(* CODESYS project vacuumsystemsimulator.library
   Title: Vacuum System Simulator Library
   Description: Library of functions used for simulation of vacuum systems.
   Placeholder: Vacuum System Simulator Library
   Version: 0.2.10
   Company: SLAC

Project tree, tasks and I/O mapping:
  libraries: Tc2_ControllerToolbox, * (Beckhoff Automation GmbH); Tc2_Standard, * (Beckhoff Automation GmbH); Tc2_System, * (Beckhoff Automation GmbH); Tc3_Interfaces, * (Beckhoff Automation GmbH); Tc3_Module, * (Beckhoff Automation GmbH)
  DUTs/
    data type ST_CapManometer
    data type ST_CapManometer_CMR362
    data type ST_GAM_PIP
    data type ST_MechPump
    data type ST_MKS_275
    data type ST_MKS_317
    data type ST_MKS_422
    data type ST_MKS_500
    data type ST_MKS_626
    data type ST_MKS_722
    data type ST_MKS_903
    data type ST_MKS_907
    data type ST_MKS_909
    data type ST_MKS_925
    data type ST_TwinScrewRoughPump
    data type ST_VacuumGauge
    data type ST_VacuumValve
    data type ST_VAT_77FS
    data type ST_Volume
  GVLs/
    global variables GVL
    global variables GVL_VSS_CONSTANT
  POUs/
    VacuumGaugePressureFunctions/
      function F_MKS_937 [ST]
    function block FB_Aperture [ST]
    function block FB_CapManometer [ST]: M_CapManometer
    function block FB_CapManometer_CMR362 [ST]: M_CapManometer_CMR362
    function block FB_GAM_PIP [ST]
    function block FB_MKS_275 [ST]
    function block FB_MKS_275_to_500_HvOn [ST]
    function block FB_MKS_422 [ST]
    function block FB_MKS_500 [ST]: M_MKS_500
    function block FB_MKS_903 [ST]: M_MKS_903
    function block FB_MKS_907 [ST]: M_MKS_907
    function block FB_MKS_909 [ST]: M_MKS_909
    function block FB_MKS_925 [ST]: M_MKS_925
    function block FB_RoughPump [ST]
    function block FB_SetChamberPressure [ST]
    function block FB_TurboPump [ST]: PumpLogic
    function block FB_VacuumValve [ST]
    function block FB_VacuumValve_Vent [ST]
    function block FB_VirtualLeak [ST]
  Version/
    global variables Global_Version
  VISUs/
*)

// DUTs/ST_CapManometer
TYPE ST_CapManometer EXTENDS ST_VacuumGauge :
STRUCT
	//rFull_Scale used for scaling the voltage range of Capacitance
	//Manometer
	rFull_Scale : REAL; //in Torr
END_STRUCT
END_TYPE

// DUTs/ST_CapManometer_CMR362
TYPE ST_CapManometer_CMR362 EXTENDS ST_VacuumGauge :
STRUCT
	(*ST_CapManometer_CMR362 is a special CapManometer with a 
	rFull_Scale = 75.0 Torr*)
	
	//rFull_Scale used for scaling the voltage range of Capacitance
	//Manometer 
	rFull_Scale : REAL := 75.0 ;// Torr
END_STRUCT
END_TYPE

// DUTs/ST_GAM_PIP
TYPE ST_GAM_PIP :
STRUCT
	//Discrete Readback 
	xOn AT%I*:BOOL; //Readback of whether Gamma Ion Pump is turned on or not
END_STRUCT
END_TYPE

// DUTs/ST_MechPump
TYPE ST_MechPump :
STRUCT
	//Simulation Parameters
	rMRE	:	REAL; // Mass Removal Efficiency: should be a number less than 1.
	rBasePress	:	REAL := 1E-3;
	rLoad	:	REAL;
	iMaxSpd	:	INT;
	rMaxLoad	:	REAL;
	tonSpd	:	TON;
	tonTemp	:	TON;
	tonOvrLd	:	TON;
	xCooling:	BOOL := FALSE; // hook the cooling active signal here
	srError	:	SR;
	rtResetErr : R_TRIG;
	
	
	//Discrete controls
	i_xIlk	:	BOOL;//allow pump to turn on
	i_xRun	:	BOOL;//actually turn on pump
	
	//Discrete readbacks
	q_xAtSpd	:	BOOL;//whether pump is at top speed
	q_xErr	:	BOOL;//whether pump has an error or faulted
	q_xStart	:	BOOL;//whether pump has started but hasnt reached top speed, returns false when reaches top speeds
	q_xLowSpd	: BOOL;//whether pump is in a lowspeed STATE
	
	//Other Readbacks
	q_iPower	:	INT;
	q_iSpeed	:	INT;
END_STRUCT
END_TYPE

// DUTs/ST_MKS_275
TYPE ST_MKS_275 EXTENDS ST_VacuumGauge :
STRUCT
	stIntrpParams	:	ST_CTRL_LIN_INTERPOLATION_PARAMS;//setup for interpolating the Pirani's funky voltage to pressure transformation
	fbInterpolator	:	FB_CTRL_LIN_INTERPOLATION := (
		bExtrapolate := TRUE //can be false too
		);
END_STRUCT
END_TYPE

// DUTs/ST_MKS_317
TYPE ST_MKS_317 EXTENDS ST_VacuumGauge :
STRUCT
END_STRUCT
END_TYPE

// DUTs/ST_MKS_422
TYPE ST_MKS_422 EXTENDS ST_VacuumGauge :
STRUCT
	
	//Discrete Control: Ion gauges only
	i_xHvOn	 AT%I*:	BOOL;//High voltage On to turn on ion gauges
	
	// Simulation parameters
	tonIC	:	TON := (PT := T#10S);// takes 10 seconds to turn on this gauge
END_STRUCT
END_TYPE

// DUTs/ST_MKS_500
TYPE ST_MKS_500 EXTENDS ST_VacuumGauge :
STRUCT
	//Discrete Control: Ion gauges only
	i_xHvOn	 AT%I*:BOOL	; //High voltage On to turn on this Cold Cathode gauge
	q_xHVOn AT%Q*:BOOL ;
	q_DisActive AT%Q*:BOOL ;
	// Simulation parameters
	tonIC	:	TON := (PT := T#10S);// takes 10 seconds to turn on this Cold Cathode gauge
END_STRUCT
END_TYPE

// DUTs/ST_MKS_626
TYPE ST_MKS_626 EXTENDS ST_VacuumGauge :
STRUCT
END_STRUCT
END_TYPE

// DUTs/ST_MKS_722
TYPE ST_MKS_722 EXTENDS ST_VacuumGauge :
STRUCT
END_STRUCT
END_TYPE

// DUTs/ST_MKS_903
TYPE ST_MKS_903 EXTENDS ST_VacuumGauge:
STRUCT

	//Discrete Control: Ion gauges only
	i_xHvOn	:	BOOL;//High voltage On to turn on this Cold Cathode gauge
	
	// Simulation parameters
	tonIC	:	TON := (PT := T#10S);// takes 10 seconds to turn on this Cold Cathode gauge

END_STRUCT
END_TYPE

// DUTs/ST_MKS_907
TYPE ST_MKS_907 EXTENDS ST_VacuumGauge :
STRUCT
	stIntrpParams	:	ST_CTRL_LIN_INTERPOLATION_PARAMS;//setup for interpolating the Pirani's funky voltage to pressure transformation
	fbInterpolator	:	FB_CTRL_LIN_INTERPOLATION := (
		bExtrapolate := FALSE
);
END_STRUCT
END_TYPE

// DUTs/ST_MKS_909
TYPE ST_MKS_909 EXTENDS ST_VacuumGauge:
STRUCT

	//Discrete Control: Ion gauges only
	i_xHvOn	:	BOOL;//High voltage On to turn on this Hot Cathode gauge, they turn on immediately, unlike cold cathodes
	
END_STRUCT
END_TYPE

// DUTs/ST_MKS_925
TYPE ST_MKS_925 EXTENDS ST_VacuumGauge :
STRUCT
END_STRUCT
END_TYPE

// DUTs/ST_TwinScrewRoughPump
TYPE ST_TwinScrewRoughPump EXTENDS ST_MechPump :
STRUCT
	//Control
	i_xLowSpd	:	BOOL;
	i_xReset	:	BOOL;
	
	//Readback
	q_xRun		:	BOOL;
	q_xStop		:	BOOL;
	
END_STRUCT
END_TYPE

// DUTs/ST_VacuumGauge
TYPE ST_VacuumGauge :
STRUCT
	(* Simulation parameters *)
	rPress	:	REAL;//The real pressure coming from the ST_volume @ a chamber
	
	(* IO Readback *)
	q_iRawPress	 AT%Q*:	INT;// The transformed integer from real pressure to an integer encoded signal to be passed to the PLC 
	
	(* Testing Connection *)
	q_xGaugeConnected	: BOOL;// to connect and disconnect gauge, easy to check whether gauge in connected at correct location

END_STRUCT
END_TYPE

// DUTs/ST_VacuumValve
TYPE ST_VacuumValve :
STRUCT

	//Discrete controls
	i_xSol	 AT%I*	:BOOL;//Solenoid to control the valve( either closed or open)
	
	//Discrete readbacks
	q_xOpnLS  AT%Q*: BOOL;//readback whether open
	q_xClsLS  AT%Q*: BOOL;//readback whether closed
END_STRUCT
END_TYPE

// DUTs/ST_VAT_77FS
TYPE ST_VAT_77FS :
STRUCT
	(*HV sensor 1*)
	q_xSens1Rdy	:	BOOL;
	q_xSens1Inrush	:	BOOL;
	i_xSens1SensorOff:	BOOL;
	
	(*HV sensor 2*)
	q_xSens2Rdy	:	BOOL;
	q_xSens2Inrush	:	BOOL;
	i_xSens2SensorOff:	BOOL;
	
	(*Control Module*)
	q_xSysRdy	:	BOOL;
	q_xClsExternal	:	BOOL;
	i_xSysReset	:	BOOL;
	
	(*Gate Module*)
	q_xGate1Open:	BOOL;
	q_xGate1Close	:	BOOL;
	q_xGate1Rdy	:	BOOL;
	
	q_xGate2Open:	BOOL;
	q_xGate2Close	:	BOOL;
	q_xGate2Rdy	:	BOOL;
	
	i_xGate1Open:	BOOL;
	i_xGate1Close	:	BOOL;
	i_xGate2Open:	BOOL;
	i_xGate2Close	:	BOOL;
	
	(*FAST Shutter Valve Module*)
	q_xFast1Rdy	:	BOOL;
	q_xFast1Inrush	:	BOOL;
	i_xFast1SensorOff:	BOOL;
	
	i_xFast1Open:	BOOL;
	i_xFast1Close	:	BOOL;

END_STRUCT
END_TYPE

// DUTs/ST_Volume
TYPE ST_Volume :
STRUCT
	(*The Volume, Pressure, and LeakRate in each chamber
	Each chamber is divided up based on the one of the pages in the drawings*)
	rVolume : REAL;	
	rPressure : REAL; //in Torr
	rVLeak	:	REAL; //Torr*L/cycle
END_STRUCT
END_TYPE

// GVLs/GVL
VAR_GLOBAL
END_VAR

// GVLs/GVL_VSS_CONSTANT
VAR_GLOBAL CONSTANT
	ATM	:	REAL := 760; // Atmospheric pressure in Torr
	tSec : INT := 1; // time in seconds
	IonMassRate : REAL := 0.00001; // Torr*Liter/seconds
END_VAR

// Version/Global_Version
{attribute 'TcGenerated'}
// This function has been automatically generated from the project information.
VAR_GLOBAL CONSTANT
	{attribute 'const_non_replaced'}
	{attribute 'linkalways'}
	stLibVersion_Vacuum_System_Simulator_Library : ST_LibVersion := (iMajor := 0, iMinor := 2, iBuild := 10, iRevision := 0, sVersion := '0.2.10');
END_VAR

// POUs/VacuumGaugePressureFunctions/F_MKS_937
FUNCTION F_MKS_937 : INT
VAR_INPUT
	rPress	:	REAL;
END_VAR
VAR
END_VAR

(* Converts real pressure to digital voltage for 937A/B *)
IF rPress <> 0 THEN
	F_MKS_937 := REAL_TO_INT( (32767/10) * (0.6* LOG( rPress ) + 7.2) );
ELSE
	F_MKS_937 := 0;
END_IF

END_FUNCTION

// POUs/FB_Aperture
FUNCTION_BLOCK FB_Aperture
VAR_INPUT
	i_rC	:	REAL := 0.5; //Conductance (less than 1)
END_VAR
VAR_OUTPUT
END_VAR
VAR_IN_OUT
	stAVol	:	ST_Volume;
	stBVol	:	ST_Volume;
END_VAR
VAR
	Pa, Va, Pb, Vb	:	REAL;
	//DeltaPa, DeltaPb	:	REAL;
END_VAR

(* Aperture Simulation
A.Pai
3/29/2017

An aperture is like a valve that is permanently open but allows a restricted
amount of mass to flow through it. It has no polarity, that is to say,
it flows the same in either direction.

An aperture is the interface between two chambers and imitates the realistic
flow rate to adjust for changing pressures
*)

// Mass flow is dependent upon pressure differential, mass flow limited by aperture size.

Pa := stAVol.rPressure;
Va := stAVol.rVolume;

Pb := stBVol.rPressure;
Vb := stBVol.rVolume;

(*simplified version of Mass in chamber = old mass - mass flow rate * time
  mass flow rate = (Pa-Pb)*(Conductance between chambers)
  mass = Pa*Va (torr * L) it should be called energy(Joules) but mass easier to visualize.
*)

stAVol.rPressure := Pa - (Pa-Pb)*i_rC*tSec/Va;
stBVol.rPressure := Pb + (Pa-Pb)*i_rC*tSec/Vb;

//need to put in when Pa== Pb and when Pa<Pb conditions

END_FUNCTION_BLOCK

// POUs/FB_CapManometer
FUNCTION_BLOCK FB_CapManometer
VAR_INPUT
	stVolume : ST_Volume;
END_VAR
VAR_OUTPUT
END_VAR
VAR_IN_OUT
	stGCM	:	ST_CapManometer;
END_VAR
VAR
END_VAR

(* 
Capacitance Manometer gauge

A Capacitance Manometer gauge takes as input, the pressure of the volume it is attached to,
and produces on its analog output, a corresponding voltage.

A. Pai, 2017-3-27
*)

IF stGCM.q_xGaugeConnected THEN//If gauge is connected

	(*set gauge real pressure based on chamber real pressure*)
	stGCM.rPress := stVolume.rPressure;
	(*set gauge raw pressure based on transformation of real pressure*)
	stGCM.q_iRawPress := M_CapManometer(stGCM);// gauge on

ELSE//gauge gets disconnected

	stGCM.rPress := 0;
	stGCM.q_iRawPress := 0; // gauge not on ??

END_IF

METHOD M_CapManometer : INT
VAR_INPUT
	stGCM	: ST_CapManometer;
END_VAR
(*
Capacitance Manometer voltage calculation 

Does the inverse of the FB_GCM from the vacuum library

A. Pai, 2017-3-27
*)
IF stGCM.rPress <> 0 THEN
	M_CapManometer := REAL_TO_INT(stGCM.rPress * 32767 / stGCM.rFull_Scale );
ELSE
	M_CapManometer := 0;
END_IF
END_METHOD

END_FUNCTION_BLOCK

// POUs/FB_CapManometer_CMR362
FUNCTION_BLOCK FB_CapManometer_CMR362
VAR_INPUT
	stVolume : ST_Volume;
END_VAR
VAR_OUTPUT
END_VAR
VAR_IN_OUT
	stGCM_362	:	ST_CapManometer_CMR362;
END_VAR
VAR
END_VAR

(* 
Capacitance Manometer gauge

A Capacitance Manometer gauge takes as input, the pressure of the volume it is attached to,
and produces on its analog output, a corresponding voltage.

A. Pai, 2017-3-27
*)

IF stGCM_362.q_xGaugeConnected THEN//If gauge is connected

	(*set gauge real pressure based on chamber real pressure*)
	stGCM_362.rPress := stVolume.rPressure;
	(*set gauge raw pressure based on transformation of real pressure*)
	stGCM_362.q_iRawPress := M_CapManometer_CMR362(stGCM_362);// gauge on

ELSE//gauge gets disconnected

	stGCM_362.rPress := 0;
	stGCM_362.q_iRawPress := 0; // gauge not on ??

END_IF

METHOD M_CapManometer_CMR362 : INT
VAR_INPUT
	stGCM_362	: ST_CapManometer_CMR362;
END_VAR
(*
Capacitance Manometer voltage calculation 

Does the inverse of the FB_GCM from the vacuum library

A. Pai, 2017-3-27
*)
IF stGCM_362.rPress <> 0 THEN
	M_CapManometer_CMR362 := REAL_TO_INT(((stGCM_362.rPress * 8 / stGCM_362.rFull_Scale) + 1)*32767/10 );
ELSE
	M_CapManometer_CMR362 := 0;
END_IF
END_METHOD

END_FUNCTION_BLOCK

// POUs/FB_GAM_PIP
FUNCTION_BLOCK FB_GAM_PIP
VAR_INPUT
END_VAR
VAR_OUTPUT
END_VAR
VAR_IN_OUT
	stVolume : ST_Volume;
	stPip	:	ST_GAM_PIP;
END_VAR
VAR
	Pa 	: REAL;
	Va	: REAL;
END_VAR

(* Ion Pump Simulation
A. Pai 2017-1-27

The Ion Pump turns gas molecules into solid by using electroplating.

Therefore the Ion Pump takes gas molecules out of the system. 
We can treat that as if a small portion of gas mass is disappearing.

*)

IF stPip.xOn THEN

Pa := stVolume.rPressure;
Va := stVolume.rVolume;
// just reduce the pressure by 0.001%
stVolume.rPressure := Pa *(0.999);

END_IF

END_FUNCTION_BLOCK

// POUs/FB_MKS_275
FUNCTION_BLOCK FB_MKS_275
VAR_INPUT
	stVolume : ST_Volume;
END_VAR
VAR_OUTPUT
END_VAR
VAR_IN_OUT
	stGauge	:	ST_MKS_275;
END_VAR
VAR
	rVoltage	:	REAL;
END_VAR
VAR CONSTANT
	caPvsV	:	ARRAY[1..31,1..2] OF LREAL := [
		0,0.375,
		1.00E-04,0.376,
		2.00E-04,0.377,
		5.00E-04,0.379,
		1.00E-03,0.384,
		2.00E-03,0.392,
		5.00E-03,0.417,
		1.00E-02,0.455,
		2.00E-02,0.523,
		5.00E-02,0.682,
		1.00E-01,0.876,
		2.00E-01,1.155,
		5.00E-01,1.683,
		1.00E+00,2.217,
		2.00E+00,2.842,
		5.00E+00,3.675,
		1.00E+01,4.206,
		2.00E+01,4.577,
		5.00E+01,4.846,
		1.00E+02,4.945,
		2.00E+02,5.019,
		3.00E+02,5.111,
		4.00E+02,5.224,
		5.00E+02,5.329,
		6.00E+02,5.419,
		7.00E+02,5.495,
		7.60E+02,5.534,
		8.00E+02,5.558,
		9.00E+02,5.614,
		1.00E+03,5.659,
		1.01E+03,5.66
	]; //the conversion table for pressure to analog (super) non-linear voltage
	caPvsVRows	:	UINT	:= 31;
END_VAR

(* 
MKS 275 Vacuum gauge

A vacuum gauge takes as input, the pressure of the volume it is attached to,
and produces on its analog output, a corresponding voltage.

A.Pai
3/29/2017
*)

(*
MKS 275 voltage calculation 

Does the inverse of the FB 275 from the vacuum library.
Converts real pressure into MKS 275 signal based on interpolation.
//not working right now
A. Pai, 2017-1-13
*)


IF stGauge.q_xGaugeConnected THEN//If gauge is connected

	(*set gauge real pressure based on chamber real pressure*)
	stGauge.rPress := stVolume.rPressure;
	(* Run the interpolator to get a new value for the analog voltage *)
	stGauge.stIntrpParams.tCtrlCycleTime := T#10MS;
	stGauge.stIntrpParams.tTaskCycleTime := T#10MS;
	stGauge.stIntrpParams.pDataTable_ADR	:=	ADR(caPvsV); //we point each time this block gets called to avoid online changes shifting memory around and potentially screwing up this pointer.
	stGauge.stIntrpParams.nDataTable_SIZEOF	:=	SIZEOF(caPvsV);
	stGauge.stIntrpParams.nDataTable_NumberOfRows := caPvsVRows;	
	
	stGauge.fbInterpolator.fIn	:=	REAL_TO_LREAL(stGauge.rPress);
	stGauge.fbInterpolator.eMode := eCTRL_MODE_ACTIVE; //active

	stGauge.fbInterpolator(stParams := stGauge.stIntrpParams, fOut => rVoltage);
	(*set gauge raw pressure based on transformation of real pressure*)
	stGauge.q_iRawPress := LREAL_TO_INT( rVoltage * 32767/10 );// gauge on

ELSE//gauge gets disconnected

	stGauge.rPress := 0;
	stGauge.q_iRawPress := 0; // gauge not on ??

END_IF

END_FUNCTION_BLOCK

// POUs/FB_MKS_275_to_500_HvOn
FUNCTION_BLOCK FB_MKS_275_to_500_HvOn
VAR_INPUT
	stPirani	:	ST_MKS_275;
END_VAR
VAR_OUTPUT
END_VAR
VAR_IN_OUT
	stCC		:	ST_MKS_500;
END_VAR
VAR
END_VAR

(* HV ON for MKS 275 Pirani Gauge to Turn on MKS 500 Cold Cathode Gauge
A. Pai 
2/8/2017


Takes in Pirani Gauge as an INPUT and Cold Cathode gauge as an IN_OUT. 
The Cold Cathode uses the Pirani Pressure to determine whether or not
to turn on or turn off. There is no turn on/ turn off timer. 
No Hysterisis either. 

Turn on timer is left to Cold Cathode Function Block.
*)
//The Cold Cathode Setpoint is 0.01 Torr

//A. Wallace, implementing hysteresis with S and R

stCC.i_xHvOn S= stPirani.rPress < 5E-3;
stCC.i_xHvOn R= stPirani.rPress >= 1.0E-2;

END_FUNCTION_BLOCK

// POUs/FB_MKS_422
FUNCTION_BLOCK FB_MKS_422
VAR_INPUT
	stVolume : ST_Volume;
END_VAR
VAR_OUTPUT
END_VAR
VAR_IN_OUT
	stGauge	:	ST_MKS_422;
END_VAR
VAR

END_VAR
VAR CONSTANT
END_VAR

(* 
MKS 422 Vacuum gauge

A vacuum gauge takes as input, the pressure of the volume it is attached to,
and produces on its analog output, a corresponding voltage.

A.Pai
3/29/2017
*)

(* Operation 
When the HV on signal is active, the gauge will take a little bit of time to
start an ion current.
*)
stGauge.tonIC.IN	:=	stGauge.i_xHvOn;	
stGauge.tonIC();


(* Pressure *)
IF stGauge.tonIC.Q AND stGauge.q_xGaugeConnected THEN//If gauge is connected and fully on

	(*set gauge real pressure based on chamber real pressure*)
	stGauge.rPress := stVolume.rPressure;
	(*set gauge raw pressure based on transformation of real pressure*)
	stGauge.q_iRawPress := F_MKS_937(stGauge.rPress);

ELSIF stGauge.i_xHvOn AND stGauge.q_xGaugeConnected THEN//If gauge is connected and starting up
	
	stGauge.rPress := 0;
	stGauge.q_iRawPress := 0; // gauge on, waiting for spark
	
ELSE//gauge gets disconnected

	stGauge.rPress := 0;
	stGauge.q_iRawPress := 0; // gauge not on

END_IF

END_FUNCTION_BLOCK

// POUs/FB_MKS_500
FUNCTION_BLOCK FB_MKS_500
VAR_INPUT
	stVolume : ST_Volume;
END_VAR
VAR_OUTPUT
END_VAR
VAR_IN_OUT
	stGauge	:	ST_MKS_500;
END_VAR
VAR
END_VAR
VAR CONSTANT
END_VAR

(* 
MKS 500 Vacuum gauge

A vacuum gauge takes as input, the pressure of the volume it is attached to,
and produces on its analog output, a corresponding voltage.

A.Pai
3/29/2017
*)

(* Operation 
When the HV on signal is active, the gauge will take a little bit of time to
start an ion current.
*)
stGauge.tonIC.IN	:=	stGauge.i_xHvOn;	
stGauge.tonIC();

stGauge.rPress := stVolume.rPressure; //always this because we assume the gauge is actually physically connected

IF stGauge.q_xGaugeConnected THEN//If gauge is connected
	
	stGauge.q_iRawPress := M_MKS_500(
	i_rPress := stGauge.rPress,
	i_xHVOn	:=	stGauge.i_xHvOn,
	i_xICOn	:=	stGauge.tonIC.Q
	);// gauge on
	
	stGauge.q_xHVOn := TRUE;
	//stGauge.i_xHvOn := TRUE;
	IF (stGauge.rPress <= 0.0001) AND (stGauge.rPress >= 1.0E-10) THEN stGauge.q_DisActive := TRUE; END_IF;

ELSE//gauge gets disconnected

	stGauge.rPress := 0;
	stGauge.q_iRawPress := 0; // gauge disconnected
	stGauge.q_xHVOn := FALSE;
	stGauge.i_xHvOn := FALSE;
	stGauge.q_DisActive := FALSE;
END_IF

METHOD PRIVATE M_MKS_500 : INT
VAR_INPUT
	i_rPress	:	REAL;
	i_xHVOn	:	BOOL;
	i_xICOn	:	BOOL;
END_VAR
VAR
	rVoltage	:	REAL;
END_VAR
VAR CONSTANT
	vBase	:	REAL := 0; //corresponding vbase 0V based on default curve.  See manual pg. 44
	pBase	:	REAL := 1.0E-10; //default curve base pressure is 1E-10. Confusing since can't actually read that low using analog out.
	vSlope	:	REAL := 1.0; //looks correct for default curve
	vNoIC	:	REAL := 0.5;
	vNoHV	:	REAL := 0.1;
END_VAR
(*
MKS 500 voltage calculation

Does the inverse of the FB 500 from the vacuum library.

A. Wallace, 2016-2-22
*)
IF i_xHVOn and i_xICOn THEN
	rVoltage := MAX(vBase, (vBase + vSlope * LOG(i_rPress/pBase)));
ELSIF i_xHVOn AND NOT i_xICOn THEN
	rVoltage := vNoIC;
ELSE
	rVoltage := vNoHV;
END_IF

M_MKS_500 := REAL_TO_INT( rVoltage * 32767/10 );
END_METHOD

END_FUNCTION_BLOCK

// POUs/FB_MKS_903
FUNCTION_BLOCK FB_MKS_903
VAR_INPUT
	stVolume : ST_Volume;
END_VAR
VAR_OUTPUT
END_VAR
VAR_IN_OUT
	stGauge	:	ST_MKS_903;
END_VAR
VAR
	dummy_WaitingForSpark : 	ST_MKS_903 := (rPress := 1E-11);
	dummy_Off		      : 	ST_MKS_903 := (rPress := 1E-4);
END_VAR

(* 
MKS 909 Vacuum gauge

A vacuum gauge takes as input, the pressure of the volume it is attached to,
and produces on its analog output, a corresponding voltage.

A.Pai
3/29/2017
*)

(* Operation 
When the HV on signal is active, the gauge will take a little bit of time to
start an ion current.
*)
stGauge.tonIC.IN	:=	stGauge.i_xHvOn;	
stGauge.tonIC();

IF stGauge.tonIC.Q AND stGauge.q_xGaugeConnected THEN//If gauge is connected and fully on

	(*set gauge real pressure based on chamber real pressure*)
	stGauge.rPress := stVolume.rPressure;
	(*set gauge raw pressure based on transformation of real pressure*)
	stGauge.q_iRawPress := M_MKS_903(stGauge);// gauge on

ELSIF stGauge.i_xHvOn AND stGauge.q_xGaugeConnected THEN//If gauge is connected and starting up

	stGauge.rPress := 0;
	stGauge.q_iRawPress := M_MKS_903(dummy_WaitingForSpark); // gauge on, waiting for spark??

ELSE//gauge gets disconnected

	stGauge.rPress := 0;
	stGauge.q_iRawPress := M_MKS_903(dummy_Off); // gauge not on??

END_IF

METHOD PRIVATE M_MKS_903 : INT
VAR_INPUT
	stGauge	: ST_MKS_903;
END_VAR
(*
MKS 903 voltage calculation 

Does the inverse of the FB 903 from the vacuum library

A. Pai, 2017-1-13
*)
IF stGauge.rPress <> 0 THEN
	M_MKS_903 := REAL_TO_INT( (32767/10) * (LOG( stGauge.rPress ) + 11) );
ELSE
	M_MKS_903 := 0;
END_IF
END_METHOD

END_FUNCTION_BLOCK

// POUs/FB_MKS_907
FUNCTION_BLOCK FB_MKS_907
VAR_INPUT
	stVolume : ST_Volume;
END_VAR
VAR_OUTPUT
END_VAR
VAR_IN_OUT
	stGauge	:	ST_MKS_907;
END_VAR
VAR
END_VAR

(* 
MKS 907 Vacuum gauge

A vacuum gauge takes as input, the pressure of the volume it is attached to,
and produces on its analog output, a corresponding voltage.

A.Pai
3/29/2017
*)

IF stGauge.q_xGaugeConnected THEN//If gauge is connected

	(*set gauge real pressure based on chamber real pressure*)
	stGauge.rPress := stVolume.rPressure;
	(*set gauge raw pressure based on transformation of real pressure*)
	stGauge.q_iRawPress := M_MKS_907(stGauge);// gauge on

ELSE//gauge gets disconnected

	stGauge.rPress := 0;
	stGauge.q_iRawPress := 0; // gauge not on ??

END_IF

METHOD PRIVATE M_MKS_907 : INT
VAR_INPUT
	stGauge	: ST_MKS_907;
END_VAR
VAR CONSTANT
	caPvsV	:	ARRAY[1..55,1..2] OF REAL := [
		1.00E-03,0.387,
		2.00E-03,0.397,
		4.00E-03,0.418,
		6.00E-03,0.437,
		8.00E-03,0.456,
		1.00E-02,0.473,
		2.00E-02,0.551,
		3.00E-02,0.619,
		4.00E-02,0.679,
		5.00E-02,0.733,
		6.00E-02,0.783,
		7.00E-02,0.830,
		8.00E-02,0.874,
		9.00E-02,0.915,		
		1.00E-01,0.955,
		2.00E-01,1.271,
		3.00E-01,1.508,
		4.00E-01,1.701,
		5.00E-01,1.864,
		6.00E-01,2.007,
		7.00E-01,2.133,
		8.00E-01,2.246,
		9.00E-01,2.348,		
		1.00E+00,2.442,
		2.00E+00,3.083,
		3.00E+00,3.452,
		4.00E+00,3.698,
		5.00E+00,3.875,
		6.00E+00,4.009,
		7.00E+00,4.114,
		8.00E+00,4.198,
		9.00E+00,4.268,		
		1.00E+01,4.327,
		2.00E+01,4.627,
		2.50E+01,4.695, 
		3.00E+01,4.743,
		4.00E+01,4.805,
		5.00E+01,4.843,
		6.00E+01,4.872,
		7.00E+01,4.891,
		7.50E+01,4.898,
		8.00E+01,4.904,
		9.00E+01,4.914,		
		1.00E+02,4.923,
		2.00E+02,4.987,
		2.50E+02,5.025, 
		3.00E+02,5.071,
		4.00E+02,5.183,
		5.00E+02,5.301,
		6.00E+02,5.397,
		7.00E+02,5.478,
		7.50E+02,5.514,
		8.00E+02,5.548,
		9.00E+02,5.610,
		1.00E+03,5.666
	]; //the conversion table for pressure to analog (super) non-linear voltage

	caPvsVRows	:	UINT	:= 55;
END_VAR
VAR
	rVoltage	:	LREAL;
END_VAR
(*
MKS 907 voltage calculation 

Does the inverse of the FB 907 from the vacuum library

A. Pai, 2017-1-13
*)

IF stGauge.rPress <> 0 THEN

	(* Run the interpolator to get a new value for the analog voltage *)
	stGauge.stIntrpParams.nDataTable_NumberOfRows := 55;
	stGauge.stIntrpParams.pDataTable_ADR	:=	ADR(caPvsV); //we point each time this block gets called to avoid online changes shifting memory around and potentially screwing up this pointer.
	stGauge.stIntrpParams.nDataTable_SIZEOF	:=	SIZEOF(caPvsV);
	stGauge.fbInterpolator.fIn	:=	stGauge.rPress;
	stGauge.fbInterpolator(stParams := stGauge.stIntrpParams, fOut => rVoltage);

	(*Calculate signal based on voltage*)
	M_MKS_907	:= LREAL_TO_INT( rVoltage * 32767/10 );

ELSE
	M_MKS_907 :=0;
END_IF
END_METHOD

END_FUNCTION_BLOCK

// POUs/FB_MKS_909
FUNCTION_BLOCK FB_MKS_909
VAR_INPUT
	stVolume : ST_Volume;
END_VAR
VAR_OUTPUT
END_VAR
VAR_IN_OUT
	stGauge	:	ST_MKS_909;
END_VAR
VAR
END_VAR

(* 
MKS 909 Vacuum gauge

A vacuum gauge takes as input, the pressure of the volume it is attached to,
and produces on its analog output, a corresponding voltage.

A.Pai
3/29/2017
*)

IF stGauge.i_xHvOn AND stGauge.q_xGaugeConnected THEN//If gauge is connected and fully on

	(*set gauge real pressure based on chamber real pressure*)
	stGauge.rPress := stVolume.rPressure;
	(*set gauge raw pressure based on transformation of real pressure*)
	stGauge.q_iRawPress := M_MKS_909(stGauge);// gauge on

ELSE//gauge gets disconnected

	stGauge.rPress := 0;
	stGauge.q_iRawPress := 0; // gauge not on ??

END_IF

METHOD PRIVATE M_MKS_909 : INT
VAR_INPUT
	stGauge	:	ST_MKS_909;
END_VAR
(* Converts real pressure to digital voltage for MKS 909 *)
IF stGauge.rPress <> 0 THEN
	M_MKS_909 := REAL_TO_INT( (32767/10) * (LOG( stGauge.rPress ) + 10) );
ELSE
	M_MKS_909 := 0;
END_IF
END_METHOD

END_FUNCTION_BLOCK

// POUs/FB_MKS_925
FUNCTION_BLOCK FB_MKS_925
VAR_INPUT
	stVolume : ST_Volume;
END_VAR
VAR_OUTPUT
END_VAR
VAR_IN_OUT
	stGauge	:	ST_MKS_925;
END_VAR
VAR
END_VAR

(* 
MKS 925 Vacuum gauge

A vacuum gauge takes as input, the pressure of the volume it is attached to,
and produces on its analog output, a corresponding voltage.

A.Pai
3/29/2017
*)

IF stGauge.q_xGaugeConnected THEN//If gauge is connected

	(*set gauge real pressure based on chamber real pressure*)
	stGauge.rPress := stVolume.rPressure;
	(*set gauge raw pressure based on transformation of real pressure*)
	stGauge.q_iRawPress := M_MKS_925(stGauge);// gauge on

ELSE//gauge gets disconnected

	stGauge.rPress := 0;
	stGauge.q_iRawPress := 0; // gauge not on ??

END_IF

METHOD PRIVATE M_MKS_925 : INT
VAR_INPUT
	stGauge	:	ST_MKS_925;
END_VAR
VAR
	rVoltage	:	REAL;
END_VAR
(*
MKS 925 voltage calculation 

Does the inverse of the FB 925 from the vacuum library

A. Pai, 2017-1-13
*)


(*Calculate signal based on voltage*)
IF stGauge.rPress <> 0 THEN
	
	(*Calculate volatage based on real pressure*)
	rVoltage:= LOG(stGauge.rPress) + 6;
	(*Calculate signal based on voltage*)
	M_MKS_925	:= REAL_TO_INT( rVoltage * 32767/10 );
	
ELSE
	M_MKS_925 := 0;
END_IF
END_METHOD

END_FUNCTION_BLOCK

// POUs/FB_RoughPump
FUNCTION_BLOCK FB_RoughPump
VAR_INPUT
END_VAR
VAR_OUTPUT
END_VAR
VAR_IN_OUT
	stVolInlet	:	ST_Volume;
	stPump	:	ST_MechPump;
END_VAR
VAR
END_VAR

(* 
Roughing pump

A roughing pump removes matter from the inlet at a specified
rate.

A. Wallace, 2016-2-28
*)

IF stPump.i_xRun THEN//Press the Pump Run button
	// drop the pressure by a small percentage of the total pressure
	stVolInlet.rPressure := MAX( stVolInlet.rPressure*(1-stPump.rMRE/stVolInlet.rVolume), stPump.rBasePress);
END_IF

END_FUNCTION_BLOCK

// POUs/FB_SetChamberPressure
FUNCTION_BLOCK FB_SetChamberPressure
VAR_IN_OUT
	chamber	: ST_Volume;
END_VAR
VAR_INPUT
	rNewPressure	: REAL;
	Override	: BOOL :=FALSE;
END_VAR
VAR_OUTPUT
END_VAR
VAR
END_VAR

//If override boolean is on then set camber pressure to new pressure
IF Override THEN
	chamber.rPressure := rNewPressure;
END_IF

END_FUNCTION_BLOCK

// POUs/FB_TurboPump
FUNCTION_BLOCK FB_TurboPump
VAR_INPUT
	RunUpTime	:	TIME := T#30S; //How long it should take for the pump to reach full speed
	OverloadTime	:	TIME := T#1S; //How long a pump will take to overload
	OverTempTime	:	TIME := T#30s; //How long a pump takes to heat up
END_VAR
VAR_IN_OUT
	stVlInlet : ST_Volume;
	stVlOutlet	:	ST_Volume;
	stPump	:	ST_MechPump;
END_VAR
VAR_OUTPUT
END_VAR
VAR
	rLoadFactor : REAL := 0.8; //
	xOverloaded	:	BOOL;
	rMaxMRR : REAL := 0.8; //arbitrary for now
	xPump	:	BOOL;
	rInletPressDelta: REAL; //Inlet pressure change in one cycle
	rMassTrans: REAL; //Mass transfered through the pump in one cycle
END_VAR

THIS^.PumpLogic();

METHOD PumpLogic : BOOL
VAR_INPUT
END_VAR
VAR
	local :BOOL;
	rSpeedFactor: REAL;
END_VAR
(*
Pfeiffer Turbo Pump

A turbo pump reduces the pressure of a volume at a certain rate, mass-removal-rate(pressure,speed,tc).
The pump does this by removing mass from the inlet volume, and transferring it to the outlet volume.
This value is linear for now, but can be calculated from a non-linear expression later...
It has a limit to how much power it can consume before causing an error.
Other limits can be programmed later, perhaps something to simulate cooling issues...

When a turbo is not spinning, it is simply a low-conductance tube. For now, we are ignoring
conductance, so we'll go ahead and say, if a turbo is not spinning, it is like an open valve...
*)
(* Pump speed *)
stPump.tonSpd.IN := xPump;
stPump.tonSpd.PT := RunUpTime; 
stPump.tonSpd(Q=>stPump.q_xAtSpd);
stPump.q_iSpeed := REAL_TO_INT(LIMIT(0,TIME_TO_REAL(stPump.tonSpd.ET)/TIME_TO_REAL(RunUpTime),1) * INT_TO_REAL(stPump.iMaxSpd) );

(* Start signal loopback *)
stPump.q_xStart := stPump.i_xRun;
IF stPump.q_xAtSpd THEN
	stPump.q_xStart := FALSE;
END_IF

(* Pump load *)
(*
We claim that pump load is a function of speed and pressure.
If the pump gets overloaded, it shuts off.
This function is a normalized measure of how loaded the pump is.
Normalized pump speed +  
Pump load is also increased by having a high foreline pressure. If the inlet pressure is low, then the foreline
pressure can be quite high, without affecting the pump too badly.
*)
//stPump.rLoad := LIMIT( 0, (INT_TO_REAL(stPump.q_iSpeed) / INT_TO_REAL(stPump.iMaxSpd)) + 
//					(stVlInlet.rPressure/ATM) - rLoadFactor, 1);
IF xPump THEN
	stPump.rLoad := LIMIT( 0, (stVlInlet.rPressure/ATM + stVlOutlet.rPressure/ATM + ( (INT_TO_REAL(stPump.iMaxSpd)- INT_TO_REAL(stPump.q_iSpeed) ) / INT_TO_REAL(stPump.iMaxSpd)))/3 , 1);
ELSE
	stPump.rLoad:= 0;
END_IF
stPump.tonOvrLd.IN := stPump.rLoad >= stPump.rMaxLoad;
stPump.tonOvrLd.PT := OverloadTime;
stPump.tonOvrLd();
xOverloaded := stPump.tonOvrLd.Q;

(* Heating up! *)
(*
You don't want to run your pump at high load for a long time, or else it will heat up and die.
If cooling is active, then the heating up threshold is raised and the time to heat overload is increased.
*)
stPump.tonTemp.PT := OverTempTime;
IF stPump.xCooling THEN
	stPump.tonTemp.PT := OverTempTime*2;
	stPump.tonTemp.IN := stPump.rLoad >= 0.8;
ELSE
	stPump.tonTemp.IN := stPump.rLoad >= 0.6;
END_IF
stPump.tonTemp();


(* Mass Removal Rate *)
(*
MRR is scaled by the current speed/ max speed. This might not be the best assumption, but it's all we got for now.
*)
stPump.rMRE := INT_TO_REAL( stPump.q_iSpeed ) /INT_TO_REAL(stPump.iMaxSpd) * rMaxMRR;

(* Error *)
(*
Your pump has pizza'd when it should've french fried...
Set error flag, reset when run goes high... for now...
*)
stPump.srError.SET1 := xOverloaded OR stPump.tonTemp.Q;
stPump.rtResetErr.CLK := stPump.i_xRun;
stPump.rtResetErr();
stPump.srError.RESET := stPump.rtResetErr.Q;
stPump.srError();
stPump.q_xErr := stPump.srError.Q1;
local :=stPump.i_xRun AND NOT stPump.q_xErr;
xPump := stPump.i_xRun AND NOT stPump.q_xErr;

(* Pumping *)
IF xPump THEN
	rInletPressDelta := stVlInlet.rPressure; //the current pressure so we can find the delta further down
	// mre should become a function of inlet and outlet pressure.
	//If the chamber pressure is lower than the pump base pressure, no pumping can occur because the mass removal efficiency effectively drops to zero.
	IF stVlInlet.rPressure > stPump.rBasePress THEN
		stVlInlet.rPressure := MAX( stPump.rBasePress, 
								stVlInlet.rPressure * (1 - stPump.rMRE/stVlInlet.rVolume) );
	END_IF
	rInletPressDelta := rInletPressDelta - stVlInlet.rPressure;
	// The total mass that was transfered through the pump
	rMassTrans	:= rInletPressDelta*stVlInlet.rVolume;
	// The outlet of the pump should be seeing whatever was removed from the inlet.
	stVlOutlet.rPressure := (rMassTrans + stVlOutlet.rPressure*stVlOutlet.rVolume)/
							(stVlOutlet.rVolume); //note, only use the outlet volume because the pump is running
ELSE //treat the pump like an open valve
	stVlOutlet.rPressure := (stVlInlet.rPressure*stVlInlet.rVolume + stVlOutlet.rPressure*stVlOutlet.rVolume)/
							(stVlInlet.rVolume+stVlOutlet.rVolume);
	stVlInlet.rPressure := stVlOutlet.rPressure; 
END_IF
END_METHOD

END_FUNCTION_BLOCK

// POUs/FB_VacuumValve
FUNCTION_BLOCK FB_VacuumValve
VAR_INPUT
	ValveTime : TIME := T#500MS;
	ETime : TIME := T#0MS;
	CalcTime : TIME := T#500MS;
END_VAR
VAR_OUTPUT
END_VAR
VAR_IN_OUT
	stAVol : ST_Volume;
	stBVol : ST_Volume;
	stValve : ST_VacuumValve;
END_VAR
VAR
	ClsTOF:TOF;
	OpnTON:TON;
	ClsInverter : BOOL;
	r_t : R_TRIG;
	f_t : F_TRIG;
	State : INT;
	//calculates prevous times to send correct PT
	CalcOpenTime : TIME := T#0MS;
		fbFirstInit : R_TRIG;
	xFirstPass	:	BOOL;

END_VAR

(* 
Vacuum Valve Simulation

A valve has two ports, A and B.
And two states, open or closed. (transition = open)
Valve open:
Average of A and B is written to both sides.

Limit switches
Solenoid goes high:
1. Normal switch goes low
2. Timer for motion elapses
3. Actuated switch goes high

Solenoid values:stValve.i_xSol
low = close valve
high = open valve

State Value:
When state = 0
	Stable state. either closed or open
When state = 1
	in the opening valve state but not fully opened
When state = 2
	in the closing valve state but not fully closed

CalcOpentime: 
	The time it takes to fully open with respect to the location of the
	valve when the solenoid changes directions, either to close or to open
	from the stable state or an inbetween state	

2017-2-17 A. Pai
*)

(*On first pass, put valve into closed valve state*)
fbFirstInit(CLK := TRUE,
			Q => xFirstPass);
IF xFirstPass THEN
	stValve.q_xClsLS := TRUE;
	stValve.q_xOpnLS := FALSE;
	State := 0;
END_IF


(* Pressure transfer *)
IF NOT stValve.q_xClsLS THEN
	stBVol.rPressure := (stAVol.rPressure*stAVol.rVolume + stBVol.rPressure*stBVol.rVolume)/(stAVol.rVolume+stBVol.rVolume);
	stAVol.rPressure := stBVol.rPressure;
END_IF

(* Valve motion *)
OpnTON.IN := stValve.i_xSol;
r_t(CLK := stValve.i_xSol); 

ClsTOF.IN := stValve.i_xSol;
f_t(CLK := stValve.i_xSol);

//If there is a rising edge then change OpnTON.PT to open valve
IF(r_t.Q)THEN
	
	IF State = 0 THEN
		
		CalcOpenTime := ValveTime;
		
	END_IF
	
	// if previous state = 2, then adjust the CalcOpenTime based on ClsTOF's elapsed time
	IF State = 2 THEN
		
		CalcOpenTime := CalcOpenTime + ClsTOF.ET;
		
	END_IF
	
	//set the Propagation time need to open the valve
	OpnTON.PT := CalcOpenTime;
	//set state = 1 for rising edge case
	State := 1;
	
END_IF

//If there is a falling edge then change ClsTOF.PT to close valve
IF(f_t.Q) THEN
	//If previous state = 0, then set CalcOpenTime to 0
	IF State = 0 THEN
		
		CalcOpenTime := T#0MS;
	
	END_IF
	
	// if previous state = 1, then adjust the CalcOpenTime based on OpnTON's elapsed time
	IF State = 1 THEN
		
		CalcOpenTime := CalcOpenTime - OpnTON.ET;
		//ClsTOF.PT := ValveTime - CalcOpenTime;
		
	END_IF
	
	//set the Propagation time need to close the valve
	ClsTOF.PT := ValveTime - CalcOpenTime;
	//set state = 2 for falling edge case
	State := 2;
	
END_IF

//run both TON and TOF timers 
OpnTON(Q=>stValve.q_xOpnLS);
ClsTOF(Q=>ClsInverter);

//Invert signal to correct value
stValve.q_xClsLS := NOT ClsInverter;

//If open and close values stablized then reset state to stable state
IF(stValve.q_xOpnLS XOR stValve.q_xClsLS) THEN
	
	// set state to STABLE state
	State := 0;
	
END_IF

END_FUNCTION_BLOCK

// POUs/FB_VacuumValve_Vent
FUNCTION_BLOCK FB_VacuumValve_Vent
VAR_INPUT
	ValveTime : TIME := T#500MS;
	ETime : TIME := T#0MS;
	CalcTime : TIME := T#500MS;
END_VAR
VAR_OUTPUT
END_VAR
VAR_IN_OUT
	stAVol : ST_Volume;
	stBVol : ST_Volume;
	stValve : ST_VacuumValve;
END_VAR
VAR
	OpnTOF:TOF;
	ClsTON:TON;
	OpnInverter : BOOL;
	r_t : R_TRIG;
	f_t : F_TRIG;
	State : INT;
	//calculates prevous times to send correct PT
	CalcOpenTime : TIME := T#0MS;
	
	fbFirstInit : R_TRIG;
	xFirstPass	:	BOOL;
END_VAR

(* 
Vacuum Vent Valve Simulation

Basically it is the opposite of the the FB_VacuumValve but the default is open instead of closed

A valve has two ports, A and B.
And 3 states:Stable(either open or closed), 1st solenoid trigger, 
consecutive solenoid triggers open or closed. 
Valve default is open:
Average of A and B is written to both sides.

Limit switches
When Solenoid goes high vent is closed:
1. Normal switch goes low
2. Timer for motion elapses
3. Actuated switch goes high

2017-2-17 A. Pai
*)

(*On first pass, put valve into closed valve state*)
fbFirstInit(CLK := TRUE,
			Q => xFirstPass);
IF xFirstPass THEN
	stValve.q_xClsLS := FALSE;
	stValve.q_xOpnLS := TRUE;
	State := 0;
END_IF

(* Pressure transfer *)
IF NOT stValve.q_xClsLS THEN
	stBVol.rPressure := (stAVol.rPressure*stAVol.rVolume + stBVol.rPressure*stBVol.rVolume)/(stAVol.rVolume+stBVol.rVolume);
	stAVol.rPressure := stBVol.rPressure;
END_IF

(* Valve motion *)
ClsTON.IN := stValve.i_xSol;
r_t(CLK := stValve.i_xSol); 

OpnTOF.IN := stValve.i_xSol;
f_t(CLK := stValve.i_xSol);

//If there is a rising edge then change ClsTON.PT to close valve
IF(r_t.Q)THEN
	IF State = 0 THEN
	CalcOpenTime := ValveTime;
	END_IF
	// if previous state = 2
	IF State = 2 THEN
		CalcOpenTime := CalcOpenTime + OpnTOF.ET;
	END_IF
	ClsTON.PT := CalcOpenTime;
	//set state = 1 for rising edge case
	State := 1;
END_IF

//If there is a falling edge then change OpnTOF.PT to open valve
IF(f_t.Q) THEN
	IF State = 0 THEN
	CalcOpenTime := T#0MS;
	END_IF
	// if previous state = 1
	IF State = 1 THEN
		CalcOpenTime := CalcOpenTime - ClsTON.ET   ;
		//OpnTOF.PT := ValveTime - CalcOpenTime;
	END_IF
	OpnTOF.PT := ValveTime - CalcOpenTime;
	//set state = 2 for falling edge case
	State := 2;
END_IF

//run both TON and TOF timers 
ClsTON(Q=>stValve.q_xClsLS);
OpnTOF(Q=>OpnInverter);

//Invert signal to correct value
stValve.q_xOpnLS := NOT OpnInverter;

//If open and close values stablized then set ETime to 0ms
IF(stValve.q_xOpnLS XOR stValve.q_xClsLS) THEN
	// reset CalcOpenTime
	//CalcOpenTime := T#0MS;
	// stable state
	State := 0;
END_IF

END_FUNCTION_BLOCK

// POUs/FB_VirtualLeak
FUNCTION_BLOCK FB_VirtualLeak
VAR_INPUT
END_VAR
VAR_IN_OUT
	stVol	:	ST_Volume;
END_VAR
VAR_OUTPUT
END_VAR
VAR
	fbRand	:	DRAND;
	lrRandomFraction: LREAL;
END_VAR

(* Virtual Leak

A virtual leak accounts for outgassing and trapped volumes in the vacuum
system. We wanted this system to be real, so we'll need virtual leaks.

Note: A virtual leak, such as this one, can also serve as a leak simulator.

This FB uses a virtual leak factor, the volume, and pressure of a vessel, to
limit a random injection of mass into the vessel.

2016-3-6, A. Wallace

*)

fbRand.Seed := 0;
fbRand(Num=>lrRandomFraction);
// The limit of virtual leaks maybe should be something less generic than atm.
stVol.rPressure := MIN( ATM, stVol.rPressure  + LREAL_TO_REAL(lrRandomFraction) * stVol.rVLeak);

END_FUNCTION_BLOCK
